FUNCTION_BLOCK FB_Cimcor_IZN10E
(*
********************************************************************************
* Name: FB_Cimcor_IZN10E
*
* Author:  Automanh
* Version: 1.0.0
*
* Description:
*  Function block for SMC IZN10E-0106 Cimcor and blow Valve
*
* Remarks:
*
* Revisions:
*   1.0 -AutomanH build
*********************************************************************************)
VAR_INPUT
 xIStart  :BOOL;//离子风棒及电磁阀启动
 xIStop		:BOOL;//离子风棒停止
 xIReset	:BOOL;//复位信号
 xICimcorMaint:BOOL;//维护信号
 xIError	:BOOL;//异常信号
 xICimcorStarted:BOOL;//离子风棒放电开始
END_VAR
VAR_OUTPUT
 xQError:BOOL;
 xQCimcorStart:BOOL;//true-离子风棒放电  false-离子风棒停止放电
 xQCimcorReset:BOOL;//复位离子风棒
 xQValveStart:BOOL;//电磁阀打开
 xQNeedMaint :BOOL;//需要维护
END_VAR
VAR
 iStartStep,iOldStartStep:INT;
 iStopStep,iOldStopStep:INT;
 iResetStep,iOldResetStep:INT;
 OperR_TRIG:ARRAY[1..4]OF R_TRIG;
 tDelay:TON;
 tTimeOut:ARRAY[1..3] OF TON;
END_VAR

ACT_Start();
ACT_Stop();
ACT_Reset();
ACT_Error();
ACT_Maint();

ACTION ACT_Error:
tTimeOut[1](IN:=  iStartStep=iOldStartStep AND iOldStartStep <>0, PT:= T#5S, Q=> , ET=> );
tTimeOut[2](IN:=  iStopStep=iOldStopStep AND iOldStopStep <>0, PT:= T#5S, Q=> , ET=> );
tTimeOut[3](IN:=  iResetStep=iOldResetStep AND iOldResetStep <>0, PT:= T#5S, Q=> , ET=> );
IF  tTimeOut[1].Q OR tTimeOut[2].Q OR  tTimeOut[3].Q OR xIError THEN
		xQError:=TRUE;
END_IF
END_ACTION

ACTION ACT_Maint:
//维护信号
IF  xICimcorMaint THEN
 	xQNeedMaint:=TRUE;
END_IF
END_ACTION

ACTION ACT_Reset:
OperR_TRIG[3](CLK:=xIReset , Q=> );
CASE iResetStep OF
 0://等待启动
 		IF  OperR_TRIG[3].Q THEN
				xIStop:=FALSE;
				xIStart:=FALSE;
				xIReset:=FALSE;
				xQError:=FALSE;
				iStartStep:=0;
				iStopStep:=0;
				iResetStep:=0;
				iResetStep:=iResetStep+1;
		END_IF
 1://复位离子封棒
 		iOldResetStep:=iResetStep;
 		xQCimcorStart:=FALSE;
		xQCimcorReset:=TRUE;
		tDelay(IN:=FALSE);
		iResetStep:=iResetStep+1;
 2://延时
 			iOldResetStep:=iResetStep;
 			tDelay(IN:= TRUE , PT:= T#200MS, Q=> , ET=> );
		IF tDelay.Q THEN
		 	iResetStep:=iResetStep+1;
			tDelay(IN:=FALSE);
		END_IF
 3://关闭复位信号
 		iOldResetStep:=iResetStep;
 		xQCimcorReset:=FALSE;
		iResetStep:=iResetStep+1;
 4://结束
 		iResetStep:=0;
END_CASE
END_ACTION

ACTION ACT_Start:
OperR_TRIG[1](CLK:=xIStart , Q=> );
CASE iStartStep OF
 0://等待启动
 		IF  OperR_TRIG[1].Q THEN
				xIStop:=FALSE;
				xIStart:=FALSE;
				iStopStep:=0;
				iStartStep:=iStartStep+1;
		END_IF
 1://开启离子风棒
 		iOldStartStep:=iStartStep;
 		xQCimcorStart:=TRUE;
		iStartStep:=iStartStep+1;
 2://检查离子风棒是否开启
 		iOldStartStep:=iStartStep;
 		IF xICimcorStarted THEN
					iStartStep:=iStartStep+1; 
		END_IF
 3://打开电磁阀
 		iOldStartStep:=iStartStep;
 		xQValveStart:=TRUE;
			iStartStep:=iStartStep+1; 
 4://结束
 		iStartStep:=0;
END_CASE
END_ACTION

ACTION ACT_Stop:
OperR_TRIG[2](CLK:=xIStop , Q=> );
CASE iStopStep OF
 0://等待启动
 		IF  OperR_TRIG[2].Q THEN
				xIStop:=FALSE;
				xIStart:=FALSE;
				iStopStep:=0;
				iStopStep:=iStopStep+1;
		END_IF
 1://关闭离子风棒
 		iOldStopStep:=iStopStep;
 		xQCimcorStart:=FALSE;
		iStopStep:=iStopStep+1;
 2://检查离子风棒是否关闭
 		iOldStopStep:=iStopStep;
 		IF  NOT xICimcorStarted THEN
					iStopStep:=iStopStep+1; 
		END_IF
 3://关闭电磁阀
 			iOldStopStep:=iStopStep;
 			xQValveStart:=FALSE;
			iStopStep:=iStopStep+1; 
 4://结束
 			iStopStep:=0;
END_CASE
END_ACTION

END_FUNCTION_BLOCK

(* stored: Version 1.1.0.1, ProductVersion 3.1.4024.9
   POU FB_Cimcor_IZN10E: Id {626a7661-cd5e-4fd6-a022-04c68b85c31b}, SpecialFunc None
   Action ACT_Error: Id {f3e34566-40ba-4e82-b133-6dd97acb1a1a}
   Action ACT_Maint: Id {fd89c97e-7b66-477c-99bf-e2acdec716a1}
   Action ACT_Reset: Id {20a6429c-89ef-4fb6-9b97-aca5c78eaaa3}
   Action ACT_Start: Id {f9e5c50e-cb1d-4284-8c5d-424f4446abd4}
   Action ACT_Stop: Id {3bcc2ad6-756c-4f66-8d45-b238523cdca7} *)
